(* LS Electric XG5000 project: FLOW_LIU *)
(* PLC LSPLC *)
(* module base 0 slot 0: Cnet:XGL-C42A/B (Cnet 통신 모듈(RS-422/485, RS-422/485)) *)
(* module base 0 slot 1: 입력 모듈:XGI-D24A/B (DC 24V 입력, 32점 (전류소스 싱크공용/ 전류소스 입력)) *)
(* module base 0 slot 2: 입력 모듈:XGI-D24A/B (DC 24V 입력, 32점 (전류소스 싱크공용/ 전류소스 입력)) *)
(* module base 0 slot 3: 출력 모듈:XGQ-TR4A/B (트랜지스터 출력, 32점 (0.1A용, 싱크출력/소스출력)) *)
(* module base 0 slot 4: 고속카운터 모듈:XGF-HO2A (고속카운터 펄스(OC) 입력형, 2채널) *)
VAR_GLOBAL
    CALCU : INT;
    COUNT_DINT : DINT;
    COUNT_INT : DINT;
    D100 : BOOL;
    INST : GET_WORD;
    INST1 : PUT_WORD;
    INST2 : PUT_INT;
    INST5 : PUT_WORD;
    SAVE : DINT;
    TOTAL : DINT;
    VALUE_HI : WORD;
    VALUE_LOW : WORD;
    _0000_CH01_NFR AT %LX60928 : BOOL; (* Cnet: New Frame Ready (Ver 6.0이상) *)
    _0004_CH0_AUXEN AT %UX0.4.371 : BOOL; (* 고속카운터 모듈: 채널0 부가기능 사용(Edge,Level)지령 *)
    _0004_CH0_AUXING AT %UX0.4.5 : BOOL; (* 고속카운터 모듈: 채널0 부가기능 동작구간표시 플래그 *)
    _0004_CH0_CNT AT %UD0.4.1 : DINT; (* 고속카운터 모듈: 채널0 현재카운트 값 *)
    _0004_CH0_CNTEN AT %UX0.4.368 : BOOL; (* 고속카운터 모듈: 채널0 카운트 동작허용(Level)지령 *)
    _0004_CH0_PREEN AT %UX0.4.369 : BOOL; (* 고속카운터 모듈: 채널0 프리셋허용(Edge) 지령 *)
    _0004_CH1_PREEN AT %UX0.4.385 : BOOL; (* 고속카운터 모듈: 채널1 프리셋 허용(Edge)지령 *)
END_VAR
VAR_GLOBAL CONSTANT
    _F0004_CH0_CNT_MODE : UINT := 00; (* 고속카운터 모듈: 채널0 카운터 종류 선택 *)
    _F0004_CH0_PRESET : UINT := 02; (* 고속카운터 모듈: 채널0 프리셋 값 설정 *)
    _F0004_CH0_REV_UNIT : UINT := 20; (* 고속카운터 모듈: 채널0 단위 시간당 회전 수 기능 1회전당 펄스 수 입력 *)
    _F0004_CH0_RPU_REAL : UINT := 192; (* 고속카운터 모듈: 채널0 단위시간당회전수 값(실수형) *)
END_VAR

(* Comments on direct variables
%MW0	HI
%MW1	LOW
*)

PROGRAM INPUT (* task: 스캔 프로그램 *)
VAR_EXTERNAL
    CALCU : INT;
    COUNT_DINT : DINT;
    COUNT_INT : DINT;
    D100 : BOOL;
    INST : GET_WORD;
    INST1 : PUT_WORD;
    INST2 : PUT_INT;
    INST5 : PUT_WORD;
    SAVE : DINT;
    TOTAL : DINT;
    VALUE_HI : WORD;
    VALUE_LOW : WORD;
    _0000_CH01_NFR : BOOL; (* AT %LX60928 *) (* Cnet: New Frame Ready (Ver 6.0이상) *)
    _0004_CH0_AUXEN : BOOL; (* AT %UX0.4.371 *) (* 고속카운터 모듈: 채널0 부가기능 사용(Edge,Level)지령 *)
    _0004_CH0_AUXING : BOOL; (* AT %UX0.4.5 *) (* 고속카운터 모듈: 채널0 부가기능 동작구간표시 플래그 *)
    _0004_CH0_CNT : DINT; (* AT %UD0.4.1 *) (* 고속카운터 모듈: 채널0 현재카운트 값 *)
    _0004_CH0_CNTEN : BOOL; (* AT %UX0.4.368 *) (* 고속카운터 모듈: 채널0 카운트 동작허용(Level)지령 *)
    _0004_CH0_PREEN : BOOL; (* AT %UX0.4.369 *) (* 고속카운터 모듈: 채널0 프리셋허용(Edge) 지령 *)
    _0004_CH1_PREEN : BOOL; (* AT %UX0.4.385 *) (* 고속카운터 모듈: 채널1 프리셋 허용(Edge)지령 *)
END_VAR
VAR
    CURRENT_GALLON : DINT;
    DONE : BOOL;
    FIN : BOOL;
    HEX : REAL;
    INST3 : TOTAL;
    INST4 : TOTAL;
    INST6 : FF;
    PRESET : BOOL;
    PRESET_PB : BOOL;
    PRESET_PB_LAMP : BOOL;
    PRESET_SIG : BOOL;
    RESET : BOOL;
    SAVE_2 : TIME;
    SAVE_AND : INT;
    START : BOOL;
    STAT : USINT;
    TOTAL_GAL : DINT;
    T_1 : BOOL;
    T_2 : BOOL;
    T_3 : BOOL;
    T_4 : BOOL;
    T_ALARM : BOOL;
    T_SAVE : INT;
    VALUE : DWORD;
    X : INT;
END_VAR
VAR_EXTERNAL CONSTANT
    _F0004_CH0_CNT_MODE : UINT; (* 고속카운터 모듈: 채널0 카운터 종류 선택 *)
    _F0004_CH0_PRESET : UINT; (* 고속카운터 모듈: 채널0 프리셋 값 설정 *)
    _F0004_CH0_REV_UNIT : UINT; (* 고속카운터 모듈: 채널0 단위 시간당 회전 수 기능 1회전당 펄스 수 입력 *)
    _F0004_CH0_RPU_REAL : UINT; (* 고속카운터 모듈: 채널0 단위시간당회전수 값(실수형) *)
END_VAR
VAR
    _e1 : R_TRIG;
    _e2 : R_TRIG;
END_VAR

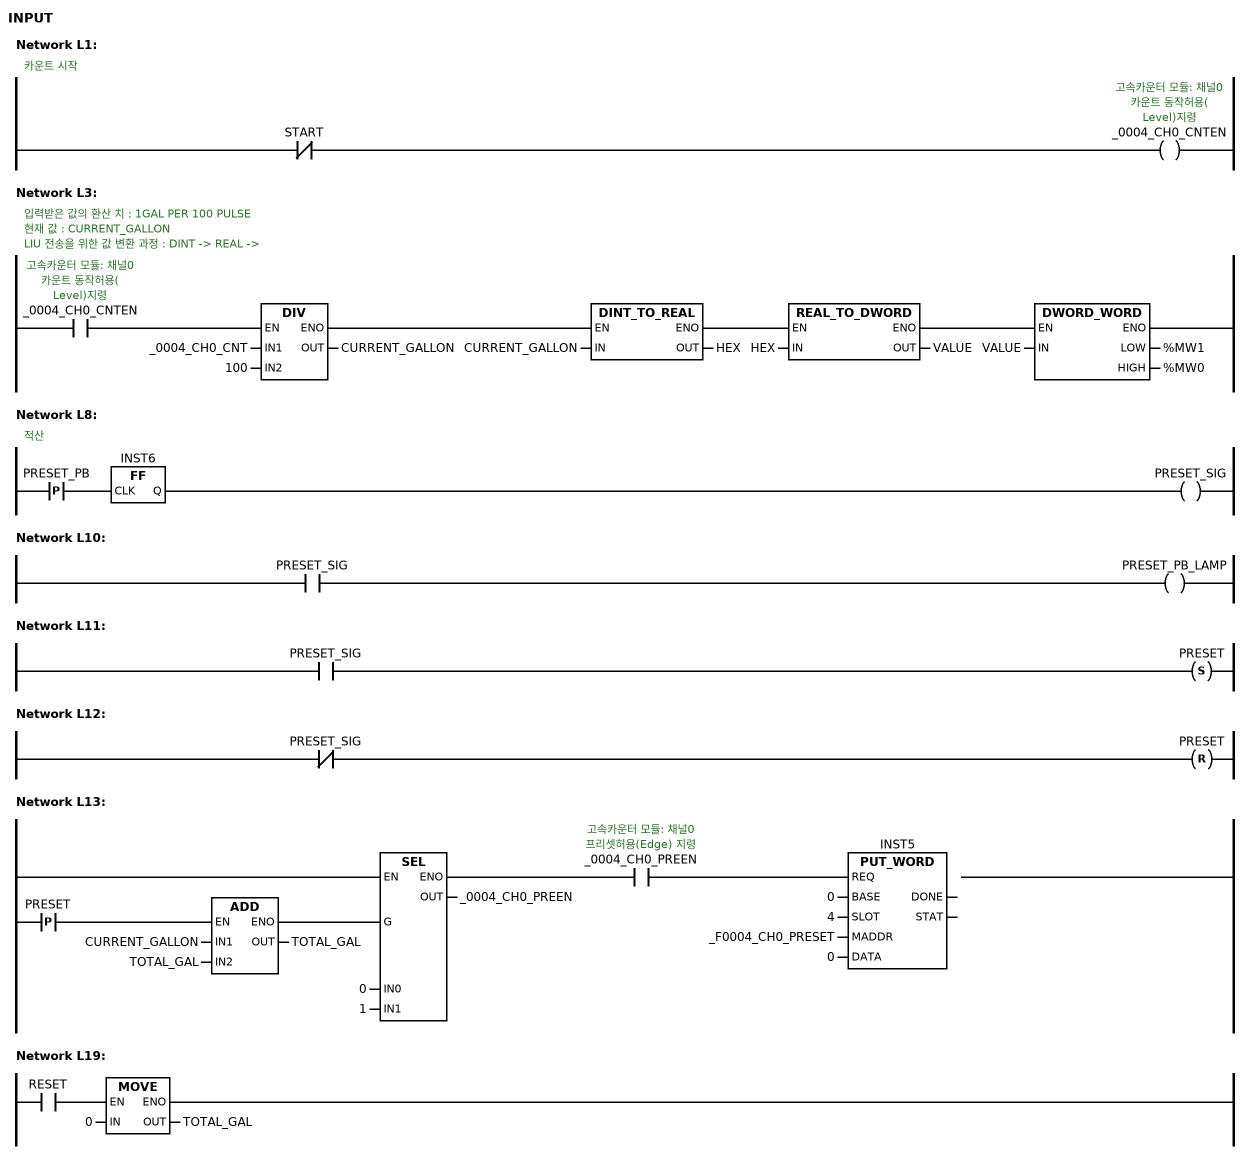
(* 카운트 시작 *)
(* Rung L1 *)
_0004_CH0_CNTEN := NOT START;
(* 입력받은 값의 환산 치 : 1GAL PER 100 PULSE / 현재 값 : CURRENT_GALLON / LIU 전송을 위한 값 변환 과정 : DINT -> REAL -> *)
(* Rung L3 *)
IF _0004_CH0_CNTEN THEN
    CURRENT_GALLON := _0004_CH0_CNT / 100;
    HEX := DINT_TO_REAL(CURRENT_GALLON);
    VALUE := REAL_TO_DWORD(HEX);
    %MW1 := DWORD_WORD(IN := VALUE, HIGH => %MW0);
END_IF;
(* 적산 *)
(* Rung L8 *)
_e1(CLK := PRESET_PB);
INST6(CLK := _e1.Q);
PRESET_SIG := INST6.Q;
(* Rung L10 *)
PRESET_PB_LAMP := PRESET_SIG;
(* Rung L11 *)
IF PRESET_SIG THEN PRESET := TRUE; END_IF;
(* Rung L12 *)
IF NOT PRESET_SIG THEN PRESET := FALSE; END_IF;
(* Rung L13 *)
_e2(CLK := PRESET);
IF _e2.Q THEN TOTAL_GAL := CURRENT_GALLON + TOTAL_GAL; END_IF;
_0004_CH0_PREEN := SEL(G := _e2.Q, IN0 := 0, IN1 := 1);
INST5(REQ := _0004_CH0_PREEN, BASE := 0, SLOT := 4, MADDR := _F0004_CH0_PRESET, DATA := 0);
(* Rung L19 *)
IF RESET THEN TOTAL_GAL := 0; END_IF;
END_PROGRAM